(* CoDeSys 2.3 export: TECHMODULE_WINDER.EXP *)
(* Libraries: 03_ApplicationModules\MPLCAxisGroupControl_Winder.lib 30.1.17 00:00:00 *)

(* Global variable list: AxisGroupControl_Winder/Version_AxisGroupControl_Winder *)
VAR_GLOBAL
	VERSION_AXISGROUPCONTROL_WINDER : DWORD := 180;
	RELEASE_AXISGROUPCONTROL_WINDER : DWORD := 100;
END_VAR

(* Global variable list: AxisGroupControl_Winder_TechModule/GlobalVar_TechModule_Winder *)
VAR_GLOBAL
{flag extrasymbolexport on}

	AxisGroupWinder		: ST_AxisGroupWinder;

{flag off}
END_VAR

VAR_GLOBAL CONSTANT
	(* Winder axis *)
	WINDER_MAX_NUMBER_OF_AXIS	:UINT:= 16;
END_VAR
